// TIA Portal V19 export
TYPE "LEXCHANGETRAY_typeConstraintWorkstationEm_recieve_interface"
// stored: Access Published
   STRUCT
      constraintRoller { S7_SetPoint := 'True'} : "LEXCHANGETRAY_typeConstraintWorkstationEm_toConstraintRollerRecieve";
   END_STRUCT;
END_TYPE
